% RSLogix 500 project training_bubble_sort_running.RSS, saved by version 8.30.00.16 %
PROJECT "UNTITLED"    % processor: Bul.1763 MicroLogix 1100 Series B %

PROGRAM FILES
  LAD 2 "MAIN"  3 rungs
  LAD 4 "LOADCELLIN"  5 rungs
  LAD 5 "TRAINING"  9 rungs
  LAD 250 "SCANHISTOG"  4 rungs
  LAD 251 "ADD_IRANK6"  7 rungs
  LAD 252 "CALC_PEAKS"  6 rungs
  LAD 253 "RNK6NEWVAL"  6 rungs
  LAD 254 "RNK6BUBBLE"  6 rungs
  LAD 255 "RESETRANK6"  5 rungs

DATA FILES
  O0 OUTPUT  4 elements
  I1 INPUT  6 elements
  S2 STATUS  66 elements
  B3 BINARY  3 elements
  T4 TIMER  2 elements
  C5 COUNTER  1 elements
  R6 CONTROL  1 elements
  N7 INTEGER  66 elements
  F8 FLOAT  1 elements
  L248 SCAN_TIMES  256 elements
  F249 RNK6FLOATS  256 elements
  N250 RNK6_INTS  256 elements
  N251 RNK6COUNTS  7 elements
  N252 RNK6BINS  7 elements
  N253 COUNT_I  256 elements
  N254 RANK6_I  256 elements
  F255 SUM_I  256 elements

LADDER 2 "MAIN"
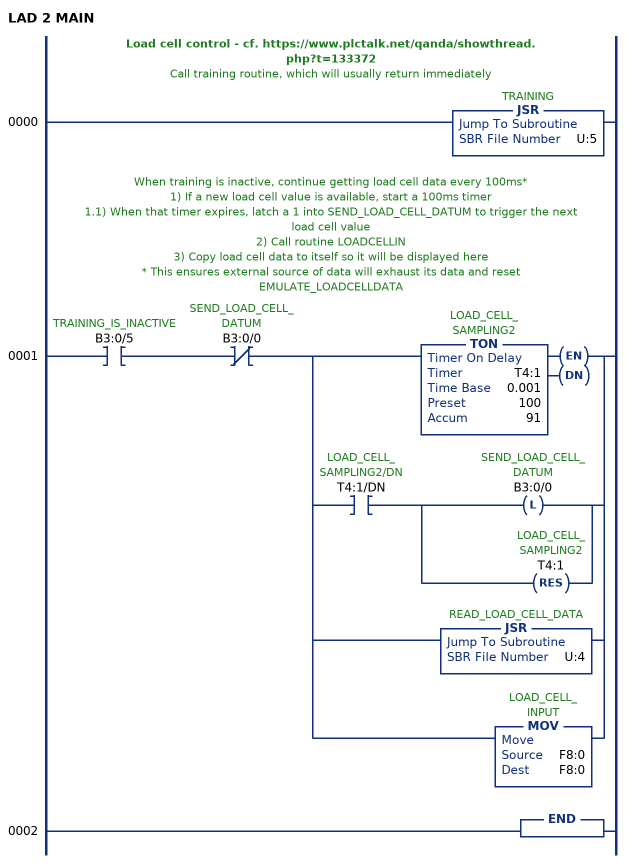
% Rung: 0 %
% TITLE: Load cell control - cf. https://www.plctalk.net/qanda/showthread.php?t=133372 %
% Call training routine, which will usually return immediately %
SOR JSR U:5 EOR
%   U:5  TRAINING %
% Rung: 1 %
% When training is inactive, continue getting load cell data every 100ms*
% 1) If a new load cell value is available, start a 100ms timer
% 1.1) When that timer expires, latch a 1 into SEND_LOAD_CELL_DATUM to trigger the next load cell value
% 2) Call routine LOADCELLIN
% 3) Copy load cell data to itself so it will be displayed here
% * This ensures external source of data will exhaust its data and reset EMULATE_LOADCELLDATA %
SOR XIC B3:0/5 XIO B3:0/0 BST BST TON T4:1 0.001 100 91 NXB XIC T4:1/DN BST OTL B3:0/0 NXB RES T4:1 BND BND NXB JSR U:4 NXB MOV F8:0 F8:0 BND EOR
%   B3:0/5  TRAINING_IS_INACTIVE %
%   B3:0/0  SEND_LOAD_CELL_DATUM %
%   T4:1  LOAD_CELL_SAMPLING2 %
%   U:4  READ_LOAD_CELL_DATA %
%   F8:0  LOAD_CELL_INPUT %
% Rung: 2 %
SOR END EOR

LADDER 4 "LOADCELLIN"
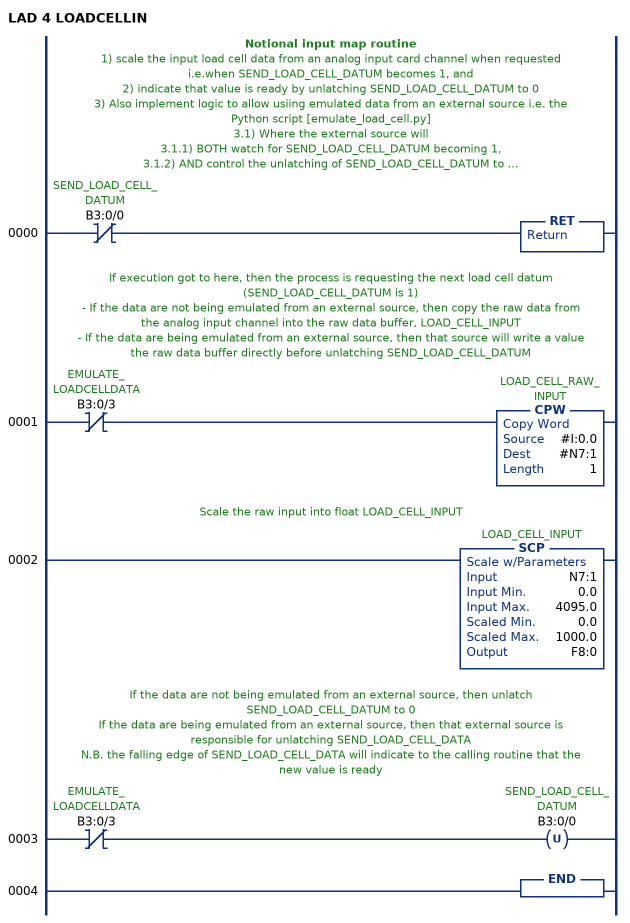
% Rung: 0 %
% TITLE: Notional input map routine %
% 1) scale the input load cell data from an analog input card channel when requested i.e.when SEND_LOAD_CELL_DATUM becomes 1, and
% 2) indicate that value is ready by unlatching SEND_LOAD_CELL_DATUM to 0
% 3) Also implement logic to allow usiing emulated data from an external source i.e. the Python script [emulate_load_cell.py]
% 3.1) Where the external source will
% 3.1.1) BOTH watch for SEND_LOAD_CELL_DATUM becoming 1,
% 3.1.2) AND control the unlatching of SEND_LOAD_CELL_DATUM to 0
% 
% ========================================================================
% If SEND_LOAD_CELL_DATA is 0 i.e. not 1, then return and do nothing %
SOR XIO B3:0/0 RET EOR
%   B3:0/0  SEND_LOAD_CELL_DATUM %
% Rung: 1 %
% If execution got to here, then the process is requesting the next load cell datum (SEND_LOAD_CELL_DATUM is 1)
% - If the data are not being emulated from an external source, then copy the raw data from the analog input channel into the raw data buffer, LOAD_CELL_INPUT
% - If the data are being emulated from an external source, then that source will write a value the raw data buffer directly before unlatching SEND_LOAD_CELL_DATUM %
SOR XIO B3:0/3 CPW #I:0.0 #N7:1 1 EOR
%   B3:0/3  EMULATE_LOADCELLDATA %
%   N7:1  LOAD_CELL_RAW_INPUT %
% Rung: 2 %
% Scale the raw input into float LOAD_CELL_INPUT %
SOR SCP N7:1 0.0 4095.0 0.0 1000.0 F8:0 EOR
%   N7:1  LOAD_CELL_RAW_INPUT %
%   F8:0  LOAD_CELL_INPUT %
% Rung: 3 %
% If the data are not being emulated from an external source, then unlatch SEND_LOAD_CELL_DATUM to 0
% If the data are being emulated from an external source, then that external source is responsible for unlatching SEND_LOAD_CELL_DATA
% N.B. the falling edge of SEND_LOAD_CELL_DATA will indicate to the calling routine that the new value is ready %
SOR XIO B3:0/3 OTU B3:0/0 EOR
%   B3:0/3  EMULATE_LOADCELLDATA %
%   B3:0/0  SEND_LOAD_CELL_DATUM %
% Rung: 4 %
SOR END EOR

LADDER 5 "TRAINING"
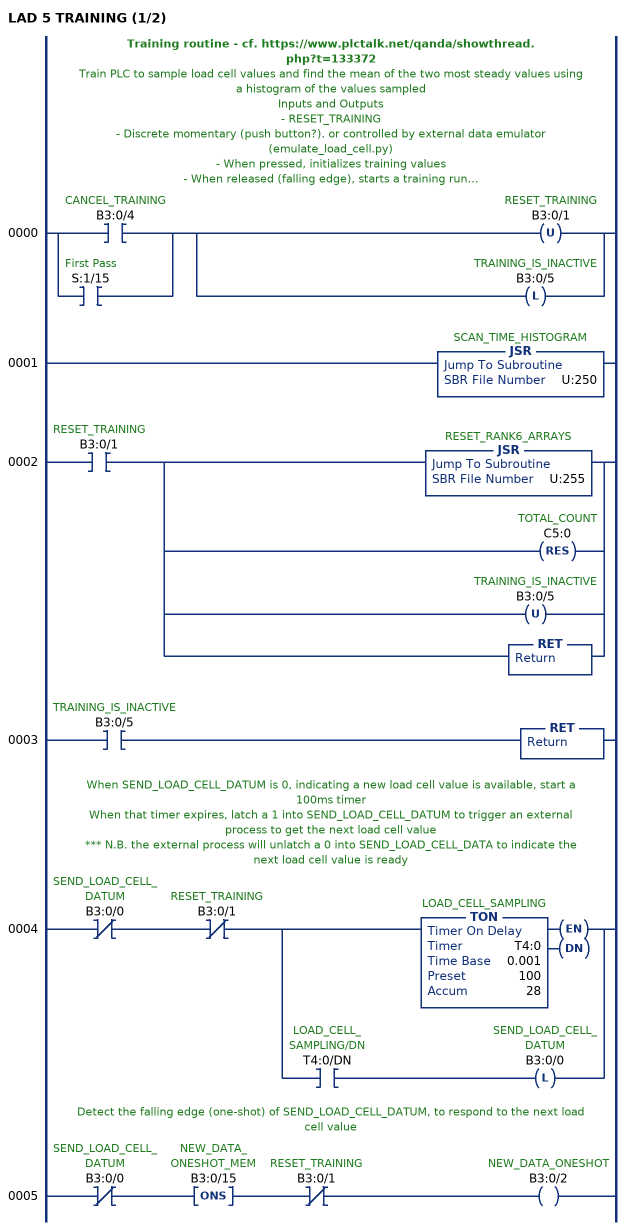
% Rung: 0 %
% TITLE: Training routine - cf. https://www.plctalk.net/qanda/showthread.php?t=133372 %
% Train PLC to sample load cell values and find the mean of the two most steady values using
% a histogram of the values sampled
% 
% Inputs and Outputs
% - RESET_TRAINING
%   - Discrete momentary (push button?). or controlled by external data emulator (emulate_load_cell.py)
%   - When pressed, initializes training values
%   - When released (falling edge), starts a training rung
% - LOAD_CELL_INPUT
%   - Analog float value that is loaded from load cell in response to a rising edge of Boolean SEND_LOAD_CELL_DATUM
% - SEND_LOAD_CELL_DATUM (both output-ish and input-ish)
%   - Output:  written to as a 1 by this routine to indicate 100ms have expired and it is time for the next load cell value
%   - Input:  written to as a 0 by another entity to after putting a new value into LOAD_CELL_INPUT
%     - This falling edge indicates a new LOAD_CELL_INPUT is ready
%     - The other entity could be an I/O mapping routine, or the Python script [emulate_load_cell.py]
% 
% ========================================================================
% First rung:  respond to request to cancel training %
SOR BST XIC B3:0/4 NXB XIC S:1/15 BND BST OTU B3:0/1 NXB OTL B3:0/5 BND EOR
%   B3:0/4  CANCEL_TRAINING %
%   S:1/15  "First Pass" %
%   B3:0/1  RESET_TRAINING %
%   B3:0/5  TRAINING_IS_INACTIVE %
% Rung: 1 %
SOR JSR U:250 EOR
%   U:250  SCAN_TIME_HISTOGRAM %
% Rung: 2 %
SOR XIC B3:0/1 BST JSR U:255 NXB RES C5:0 NXB OTU B3:0/5 NXB RET BND EOR
%   B3:0/1  RESET_TRAINING %
%   U:255  RESET_RANK6_ARRAYS %
%   C5:0  TOTAL_COUNT %
%   B3:0/5  TRAINING_IS_INACTIVE %
% Rung: 3 %
SOR XIC B3:0/5 RET EOR
%   B3:0/5  TRAINING_IS_INACTIVE %
% Rung: 4 %
% When SEND_LOAD_CELL_DATUM is 0, indicating a new load cell value is available, start a 100ms timer
% When that timer expires, latch a 1 into SEND_LOAD_CELL_DATUM to trigger an external process to get the next load cell value
% *** N.B. the external process will unlatch a 0 into SEND_LOAD_CELL_DATA to indicate the next load cell value is ready %
SOR XIO B3:0/0 XIO B3:0/1 BST TON T4:0 0.001 100 28 NXB XIC T4:0/DN OTL B3:0/0 BND EOR
%   B3:0/0  SEND_LOAD_CELL_DATUM %
%   B3:0/1  RESET_TRAINING %
%   T4:0  LOAD_CELL_SAMPLING %
% Rung: 5 %
% Detect the falling edge (one-shot) of SEND_LOAD_CELL_DATUM, to respond to the next load cell value %
SOR XIO B3:0/0 ONS B3:0/15 XIO B3:0/1 OTE B3:0/2 EOR
%   B3:0/0  SEND_LOAD_CELL_DATUM %
%   B3:0/15  NEW_DATA_ONESHOT_MEM %
%   B3:0/1  RESET_TRAINING %
%   B3:0/2  NEW_DATA_ONESHOT %

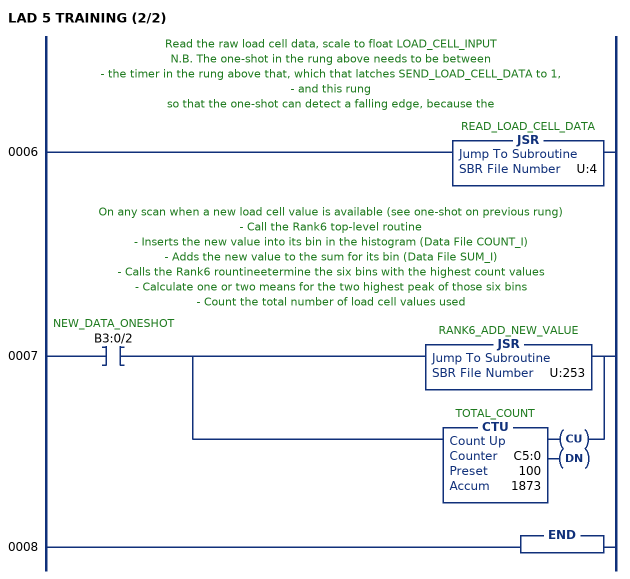
% Rung: 6 %
% Read the raw load cell data, scale to float LOAD_CELL_INPUT
% 
% N.B. The one-shot in the rung above needs to be between
%         - the timer in the rung above that, which that latches SEND_LOAD_CELL_DATA to 1,
%         - and this rung
%         so that the one-shot can detect a falling edge, because the %
SOR JSR U:4 EOR
%   U:4  READ_LOAD_CELL_DATA %
% Rung: 7 %
% On any scan when a new load cell value is available (see one-shot on previous rung)
% - Call the Rank6 top-level routine
%   - Inserts the new value into its bin in the histogram (Data File COUNT_I)
%   - Adds the new value to the sum for its bin (Data File SUM_I)
%   - Calls the Rank6 rountineetermine the six bins with the highest count values
%   - Calculate one or two means for the two highest peak of those six bins
% - Count the total number of load cell values used %
SOR XIC B3:0/2 BST JSR U:253 NXB CTU C5:0 100 1873 BND EOR
%   B3:0/2  NEW_DATA_ONESHOT %
%   U:253  RANK6_ADD_NEW_VALUE %
%   C5:0  TOTAL_COUNT %
% Rung: 8 %
SOR END EOR

LADDER 250 "SCANHISTOG"
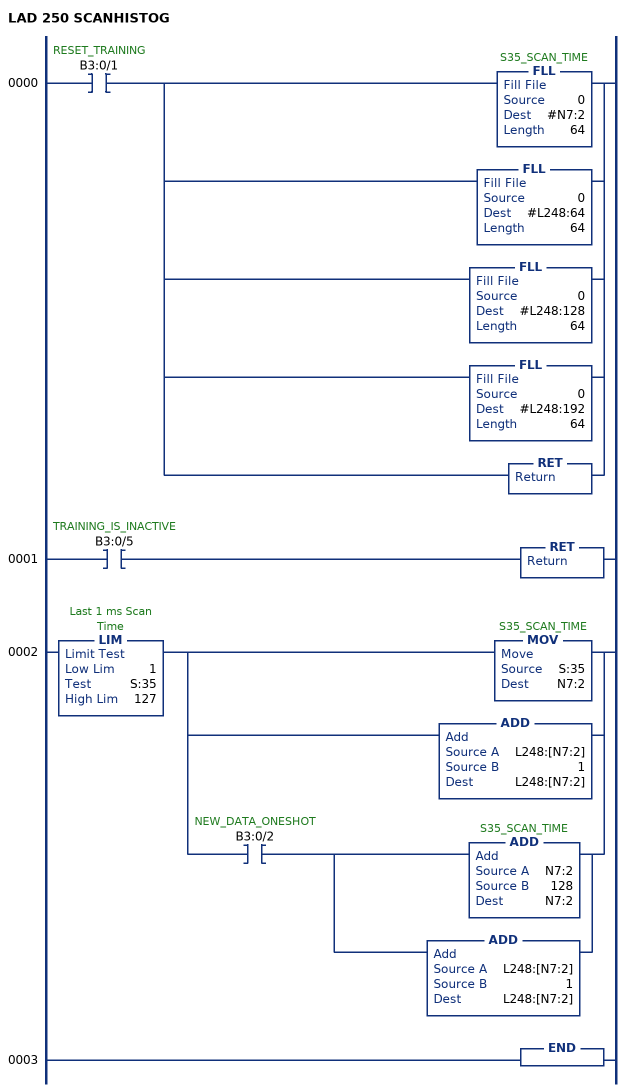
% Rung: 0 %
SOR XIC B3:0/1 BST FLL 0 #N7:2 64 NXB FLL 0 #L248:64 64 NXB FLL 0 #L248:128 64 NXB FLL 0 #L248:192 64 NXB RET BND EOR
%   B3:0/1  RESET_TRAINING %
%   N7:2  S35_SCAN_TIME %
% Rung: 1 %
SOR XIC B3:0/5 RET EOR
%   B3:0/5  TRAINING_IS_INACTIVE %
% Rung: 2 %
SOR LIM 1 S:35 127 BST MOV S:35 N7:2 NXB ADD L248:[N7:2] 1 L248:[N7:2] NXB XIC B3:0/2 BST ADD N7:2 128 N7:2 NXB ADD L248:[N7:2] 1 L248:[N7:2] BND BND EOR
%   S:35  "Last 1 ms Scan Time" %
%   N7:2  S35_SCAN_TIME %
%   B3:0/2  NEW_DATA_ONESHOT %
% Rung: 3 %
SOR END EOR

LADDER 251 "ADD_IRANK6"
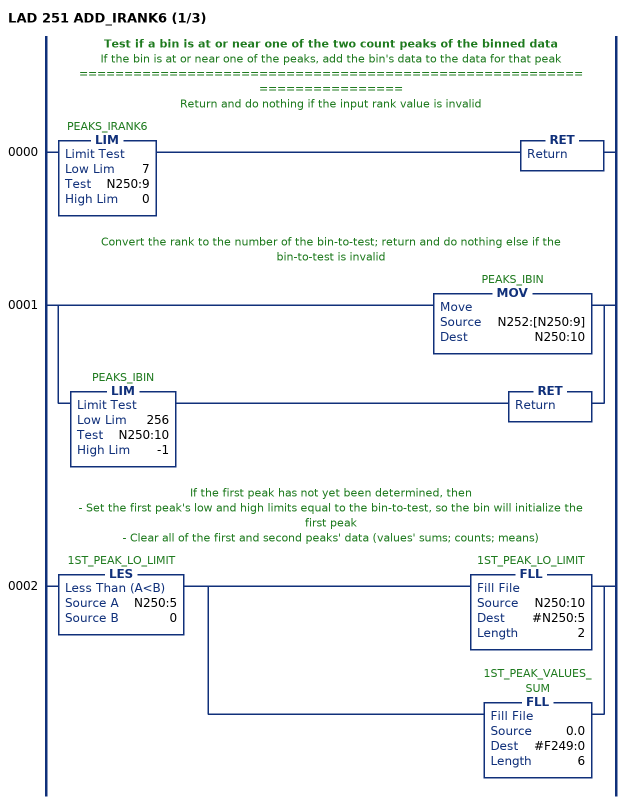
% Rung: 0 %
% TITLE: Test if a bin is at or near one of the two count peaks of the binned data %
% If the bin is at or near one of the peaks, add the bin's data to the data for that peak
% 
% ========================================================================
% Return and do nothing if the input rank value is invalid %
SOR LIM 7 N250:9 0 RET EOR
%   N250:9  PEAKS_IRANK6 %
% Rung: 1 %
% Convert the rank to the number of the bin-to-test; return and do nothing else if the bin-to-test is invalid %
SOR BST MOV N252:[N250:9] N250:10 NXB LIM 256 N250:10 -1 RET BND EOR
%   N250:9  PEAKS_IRANK6 %
%   N250:10  PEAKS_IBIN %
% Rung: 2 %
% If the first peak has not yet been determined, then
% - Set the first peak's low and high limits equal to the bin-to-test, so the bin will initialize the first peak
% - Clear all of the first and second peaks' data (values' sums; counts; means) %
SOR LES N250:5 0 BST FLL N250:10 #N250:5 2 NXB FLL 0.0 #F249:0 6 BND EOR
%   N250:5  1ST_PEAK_LO_LIMIT %
%   N250:10  PEAKS_IBIN %
%   F249:0  1ST_PEAK_VALUES_SUM %

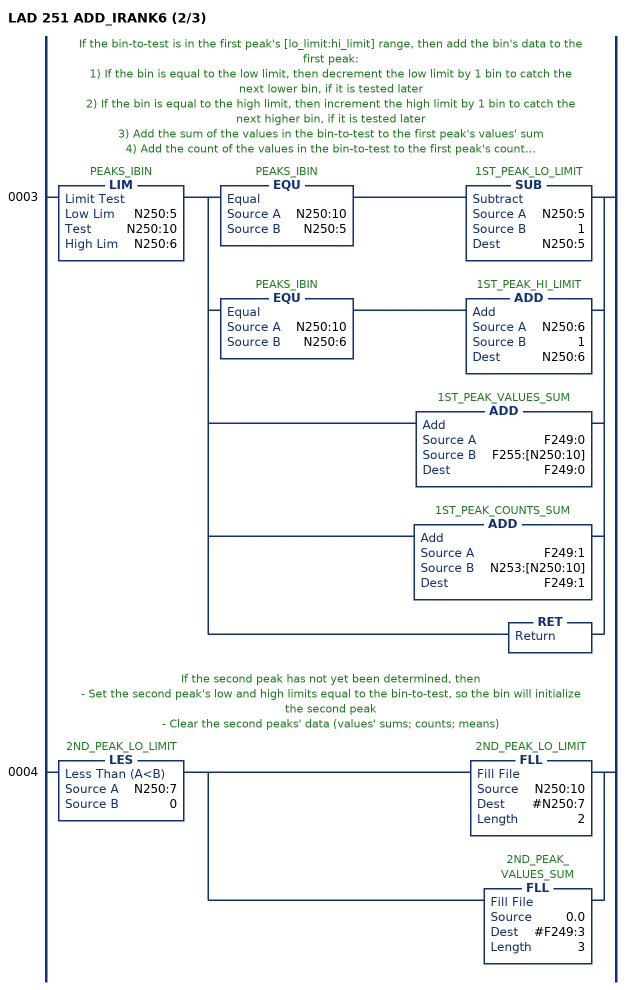
% Rung: 3 %
% If the bin-to-test is in the first peak's [lo_limit:hi_limit] range, then add the bin's data to the first peak:
% 1) If the bin is equal to the low limit, then decrement the low limit by 1 bin to catch the next lower bin, if it is tested later
% 2) If the bin is equal to the high limit, then increment the high limit by 1 bin to catch the next higher bin, if it is tested later
% 3) Add the sum of the values in the bin-to-test to the first peak's values' sum
% 4) Add the count of the values in the bin-to-test to the first peak's counts
% 5) Return and do nothing else in this routine, because the bin-to-test is in the first peak, so it cannot be in the second peak %
SOR LIM N250:5 N250:10 N250:6 BST EQU N250:10 N250:5 SUB N250:5 1 N250:5 NXB EQU N250:10 N250:6 ADD N250:6 1 N250:6 NXB ADD F249:0 F255:[N250:10] F249:0 NXB ADD F249:1 N253:[N250:10] F249:1 NXB RET BND EOR
%   N250:5  1ST_PEAK_LO_LIMIT %
%   N250:10  PEAKS_IBIN %
%   N250:6  1ST_PEAK_HI_LIMIT %
%   F249:0  1ST_PEAK_VALUES_SUM %
%   F249:1  1ST_PEAK_COUNTS_SUM %
% Rung: 4 %
% If the second peak has not yet been determined, then
% - Set the second peak's low and high limits equal to the bin-to-test, so the bin will initialize the second peak
% - Clear the second peaks' data (values' sums; counts; means) %
SOR LES N250:7 0 BST FLL N250:10 #N250:7 2 NXB FLL 0.0 #F249:3 3 BND EOR
%   N250:7  2ND_PEAK_LO_LIMIT %
%   N250:10  PEAKS_IBIN %
%   F249:3  2ND_PEAK_VALUES_SUM %

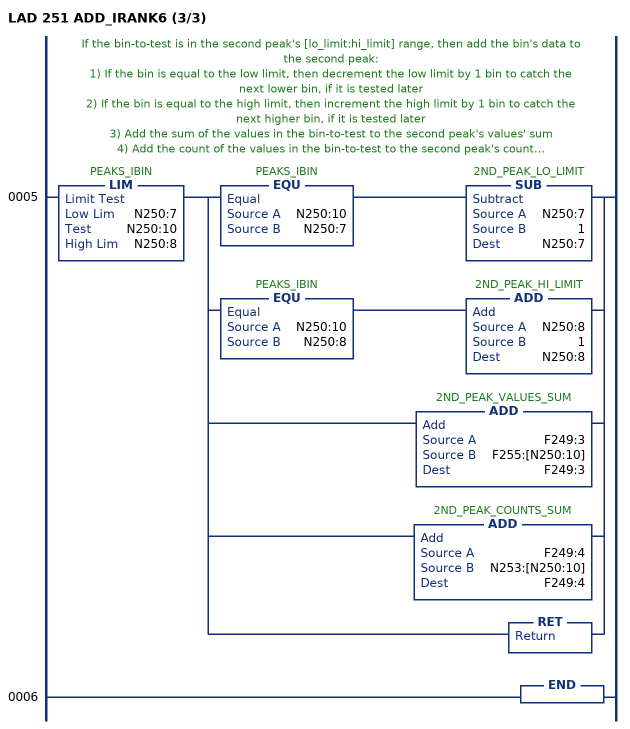
% Rung: 5 %
% If the bin-to-test is in the second peak's [lo_limit:hi_limit] range, then add the bin's data to the second peak:
% 1) If the bin is equal to the low limit, then decrement the low limit by 1 bin to catch the next lower bin, if it is tested later
% 2) If the bin is equal to the high limit, then increment the high limit by 1 bin to catch the next higher bin, if it is tested later
% 3) Add the sum of the values in the bin-to-test to the second peak's values' sum
% 4) Add the count of the values in the bin-to-test to the second peak's counts
% 5) The return is superfluous since this was originally the last rung in this routine, but this leaves open the possibility to add more peaks %
SOR LIM N250:7 N250:10 N250:8 BST EQU N250:10 N250:7 SUB N250:7 1 N250:7 NXB EQU N250:10 N250:8 ADD N250:8 1 N250:8 NXB ADD F249:3 F255:[N250:10] F249:3 NXB ADD F249:4 N253:[N250:10] F249:4 NXB RET BND EOR
%   N250:7  2ND_PEAK_LO_LIMIT %
%   N250:10  PEAKS_IBIN %
%   N250:8  2ND_PEAK_HI_LIMIT %
%   F249:3  2ND_PEAK_VALUES_SUM %
%   F249:4  2ND_PEAK_COUNTS_SUM %
% Rung: 6 %
SOR END EOR

LADDER 252 "CALC_PEAKS"
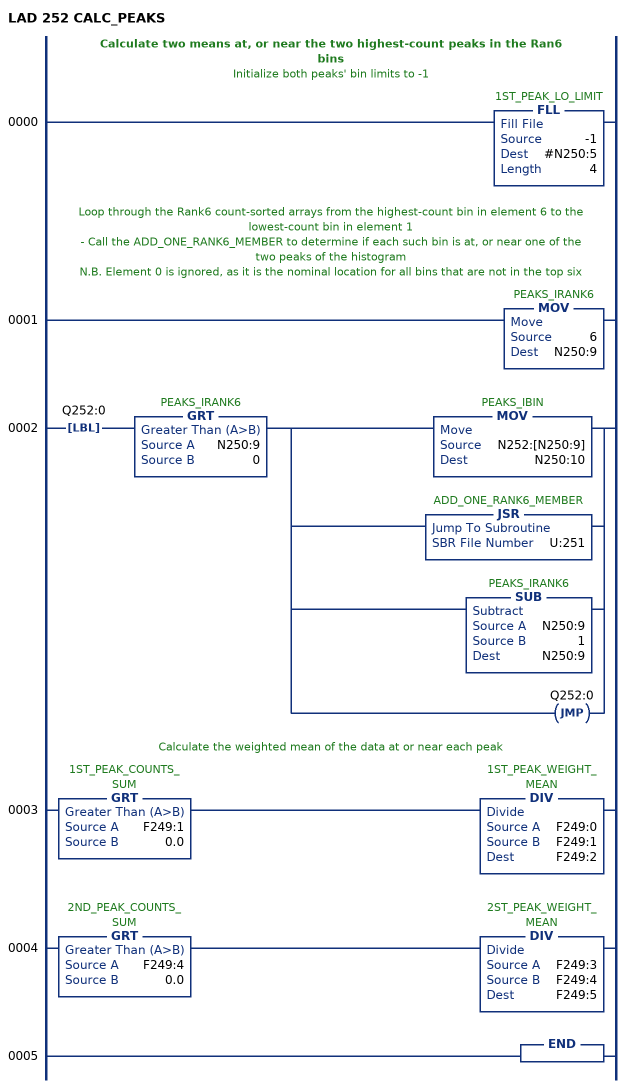
% Rung: 0 %
% TITLE: Calculate two means at, or near the two highest-count peaks in the Ran6 bins %
% Initialize both peaks' bin limits to -1 %
SOR FLL -1 #N250:5 4 EOR
%   N250:5  1ST_PEAK_LO_LIMIT %
% Rung: 1 %
% Loop through the Rank6 count-sorted arrays from the highest-count bin in element 6 to the lowest-count bin in element 1
% - Call the ADD_ONE_RANK6_MEMBER to determine if each such bin is at, or near one of the two peaks of the histogram
% N.B. Element 0 is ignored, as it is the nominal location for all bins that are not in the top six %
SOR MOV 6 N250:9 EOR
%   N250:9  PEAKS_IRANK6 %
% Rung: 2 %
SOR LBL Q252:0 GRT N250:9 0 BST MOV N252:[N250:9] N250:10 NXB JSR U:251 NXB SUB N250:9 1 N250:9 NXB JMP Q252:0 BND EOR
%   N250:9  PEAKS_IRANK6 %
%   N250:10  PEAKS_IBIN %
%   U:251  ADD_ONE_RANK6_MEMBER %
% Rung: 3 %
% Calculate the weighted mean of the data at or near each peak %
SOR GRT F249:1 0.0 DIV F249:0 F249:1 F249:2 EOR
%   F249:1  1ST_PEAK_COUNTS_SUM %
%   F249:0  1ST_PEAK_VALUES_SUM %
%   F249:2  1ST_PEAK_WEIGHT_MEAN %
% Rung: 4 %
SOR GRT F249:4 0.0 DIV F249:3 F249:4 F249:5 EOR
%   F249:4  2ND_PEAK_COUNTS_SUM %
%   F249:3  2ND_PEAK_VALUES_SUM %
%   F249:5  2ST_PEAK_WEIGHT_MEAN %
% Rung: 5 %
SOR END EOR

LADDER 253 "RNK6NEWVAL"
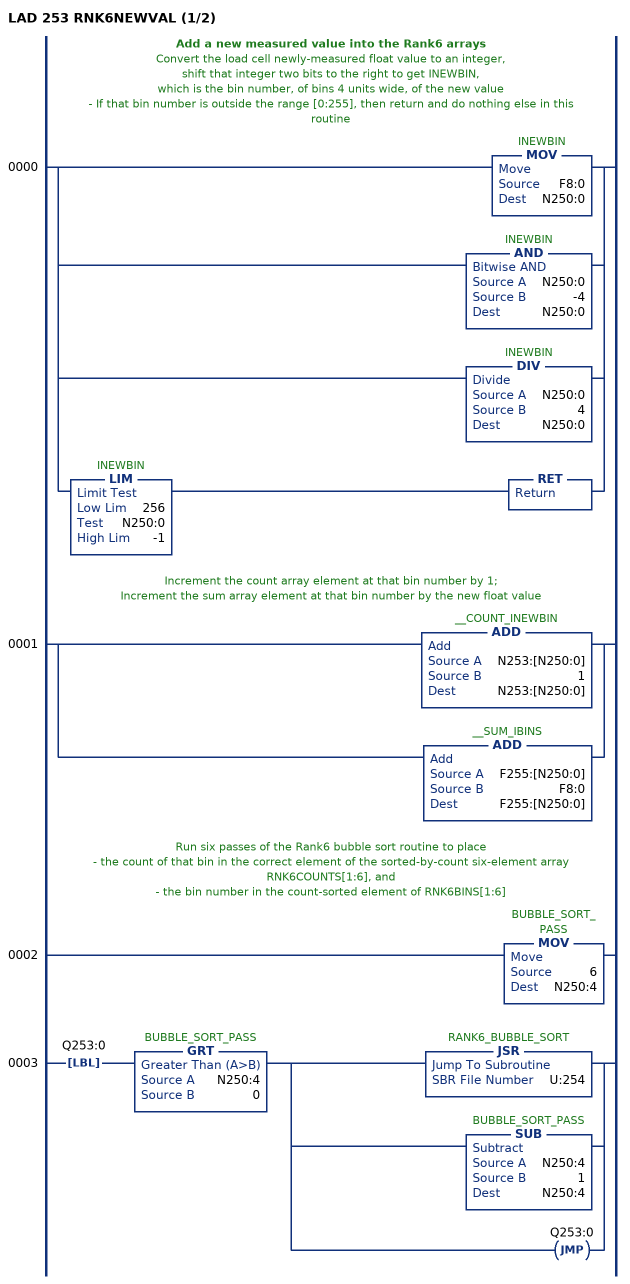
% Rung: 0 %
% TITLE: Add a new measured value into the Rank6 arrays %
% Convert the load cell newly-measured float value to an integer,
% shift that integer two bits to the right to get INEWBIN,
% which is the bin number, of bins 4 units wide, of the new value
% - If that bin number is outside the range [0:255], then return and do nothing else in this routine %
SOR BST MOV F8:0 N250:0 NXB AND N250:0 -4 N250:0 NXB DIV N250:0 4 N250:0 NXB LIM 256 N250:0 -1 RET BND EOR
%   F8:0  LOAD_CELL_INPUT %
%   N250:0  INEWBIN %
% Rung: 1 %
% Increment the count array element at that bin number by 1;
% Increment the sum array element at that bin number by the new float value %
SOR BST ADD N253:[N250:0] 1 N253:[N250:0] NXB ADD F255:[N250:0] F8:0 F255:[N250:0] BND EOR
%   N253:[N250:0]  __COUNT_INEWBIN %
%   N250:0  INEWBIN %
%   F255:[N250:0]  __SUM_IBINS %
%   F8:0  LOAD_CELL_INPUT %
% Rung: 2 %
% Run six passes of the Rank6 bubble sort routine to place
% - the count of that bin in the correct element of the sorted-by-count six-element array RNK6COUNTS[1:6], and
% - the bin number in the count-sorted element of RNK6BINS[1:6] %
SOR MOV 6 N250:4 EOR
%   N250:4  BUBBLE_SORT_PASS %
% Rung: 3 %
SOR LBL Q253:0 GRT N250:4 0 BST JSR U:254 NXB SUB N250:4 1 N250:4 NXB JMP Q253:0 BND EOR
%   N250:4  BUBBLE_SORT_PASS %
%   U:254  RANK6_BUBBLE_SORT %

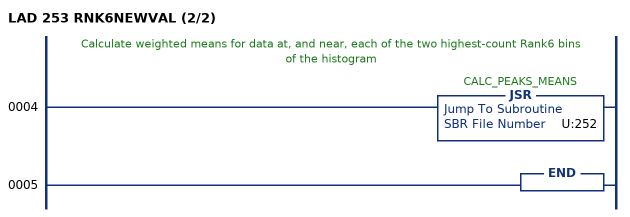
% Rung: 4 %
% Calculate weighted means for data at, and near, each of the two highest-count Rank6 bins of the histogram %
SOR JSR U:252 EOR
%   U:252  CALC_PEAKS_MEANS %
% Rung: 5 %
SOR END EOR

LADDER 254 "RNK6BUBBLE"
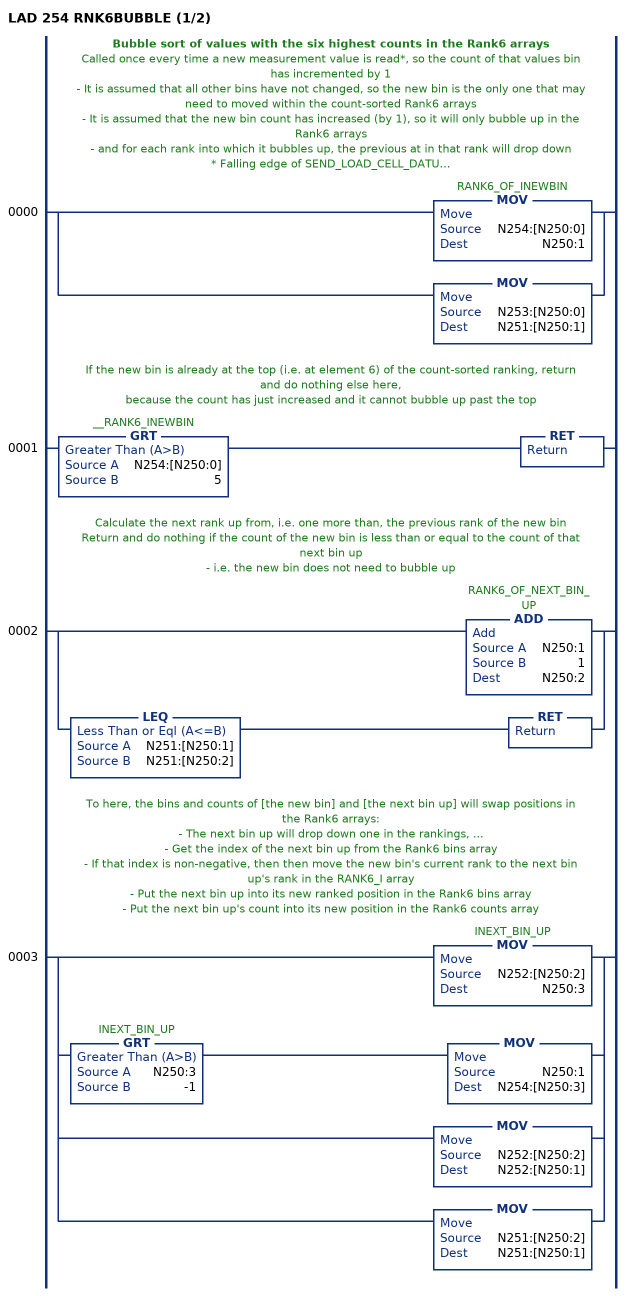
% Rung: 0 %
% TITLE: Bubble sort of values with the six highest counts in the Rank6 arrays %
% Called once every time a new measurement value is read*, so the count of that values bin has incremented by 1
% - It is assumed that all other bins have not changed, so the new bin is the only one that may need to moved within the count-sorted Rank6 arrays
% - It is assumed that the new bin count has increased (by 1), so it will only bubble up in the Rank6 arrays
%   - and for each rank into which it bubbles up, the previous at in that rank will drop down
% 
% * Falling edge of SEND_LOAD_CELL_DATUM
% 
% ========================================================================
% Get current rank of the new bin from the Rank6 bins array
% Place the updated count of the new bin in the ranked position of that bin in the Rank6 counts array %
SOR BST MOV N254:[N250:0] N250:1 NXB MOV N253:[N250:0] N251:[N250:1] BND EOR
%   N254:[N250:0]  __RANK6_INEWBIN %
%   N250:0  INEWBIN %
%   N250:1  RANK6_OF_INEWBIN %
%   N253:[N250:0]  __COUNT_INEWBIN %
% Rung: 1 %
% If the new bin is already at the top (i.e. at element 6) of the count-sorted ranking, return and do nothing else here,
% because the count has just increased and it cannot bubble up past the top %
SOR GRT N254:[N250:0] 5 RET EOR
%   N254:[N250:0]  __RANK6_INEWBIN %
%   N250:0  INEWBIN %
% Rung: 2 %
% Calculate the next rank up from, i.e. one more than, the previous rank of the new bin
% Return and do nothing if the count of the new bin is less than or equal to the count of that next bin up
% - i.e. the new bin does not need to bubble up %
SOR BST ADD N250:1 1 N250:2 NXB LEQ N251:[N250:1] N251:[N250:2] RET BND EOR
%   N250:1  RANK6_OF_INEWBIN %
%   N250:2  RANK6_OF_NEXT_BIN_UP %
% Rung: 3 %
% To here, the bins and counts of [the new bin] and [the next bin up] will swap positions in the Rank6 arrays:
% - The next bin up will drop down one in the rankings, ...
%   - Get the index of the next bin up from the Rank6 bins array
%   - If that index is non-negative, then then move the new bin's current rank to the next bin up's rank in the RANK6_I array
%   - Put the next bin up into its new ranked position in the Rank6 bins array
%   - Put the next bin up's count into its new position in the Rank6 counts array %
SOR BST MOV N252:[N250:2] N250:3 NXB GRT N250:3 -1 MOV N250:1 N254:[N250:3] NXB MOV N252:[N250:2] N252:[N250:1] NXB MOV N251:[N250:2] N251:[N250:1] BND EOR
%   N250:2  RANK6_OF_NEXT_BIN_UP %
%   N250:3  INEXT_BIN_UP %
%   N250:1  RANK6_OF_INEWBIN %

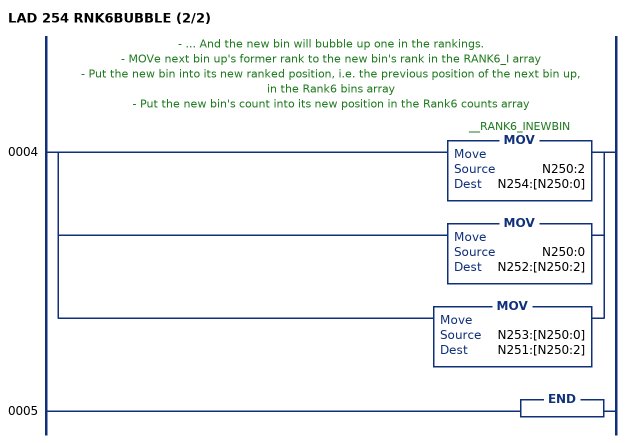
% Rung: 4 %
% - ... And the new bin will bubble up one in the rankings.
%   - MOVe next bin up's former rank to the new bin's rank in the RANK6_I array
%   - Put the new bin into its new ranked position, i.e. the previous position of the next bin up, in the Rank6 bins array
%   - Put the new bin's count into its new position in the Rank6 counts array %
SOR BST MOV N250:2 N254:[N250:0] NXB MOV N250:0 N252:[N250:2] NXB MOV N253:[N250:0] N251:[N250:2] BND EOR
%   N250:2  RANK6_OF_NEXT_BIN_UP %
%   N254:[N250:0]  __RANK6_INEWBIN %
%   N250:0  INEWBIN %
%   N253:[N250:0]  __COUNT_INEWBIN %
% Rung: 5 %
SOR END EOR

LADDER 255 "RESETRANK6"
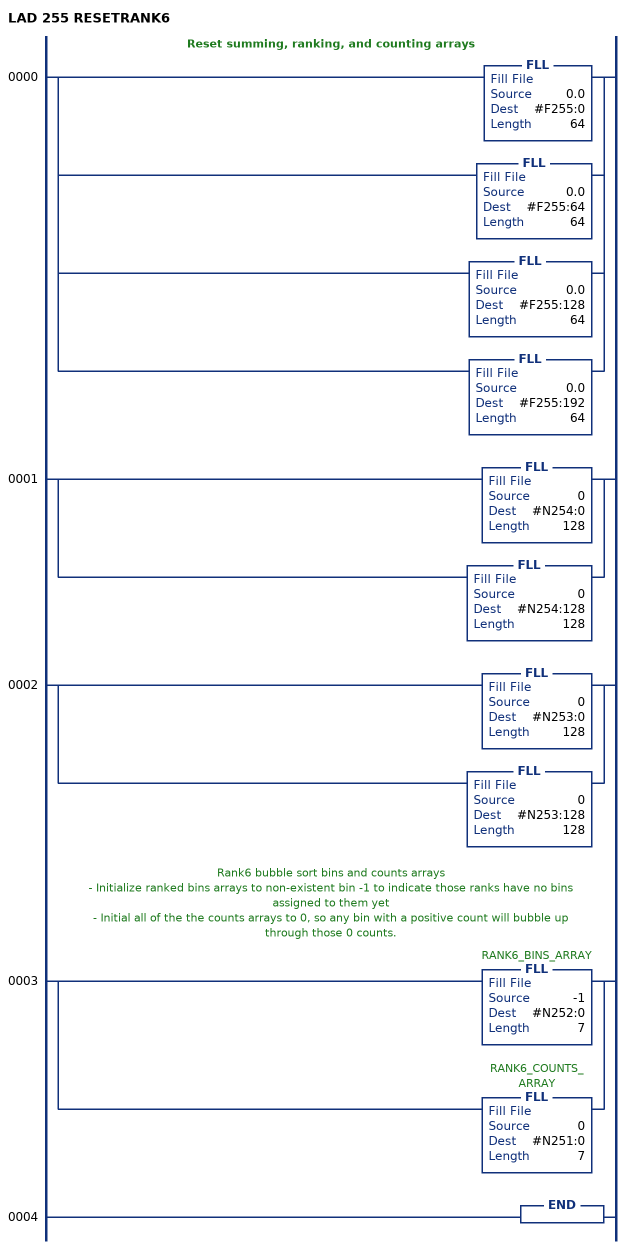
% Rung: 0 %
% TITLE: Reset summing, ranking, and counting arrays %
SOR BST FLL 0.0 #F255:0 64 NXB FLL 0.0 #F255:64 64 NXB FLL 0.0 #F255:128 64 NXB FLL 0.0 #F255:192 64 BND EOR
% Rung: 1 %
SOR BST FLL 0 #N254:0 128 NXB FLL 0 #N254:128 128 BND EOR
% Rung: 2 %
SOR BST FLL 0 #N253:0 128 NXB FLL 0 #N253:128 128 BND EOR
% Rung: 3 %
% Rank6 bubble sort bins and counts arrays
% - Initialize ranked bins arrays to non-existent bin -1 to indicate those ranks have no bins assigned to them yet
% - Initial all of the the counts arrays to 0, so any bin with a positive count will bubble up through those 0 counts. %
SOR BST FLL -1 #N252:0 7 NXB FLL 0 #N251:0 7 BND EOR
%   N252:0  RANK6_BINS_ARRAY %
%   N251:0  RANK6_COUNTS_ARRAY %
% Rung: 4 %
SOR END EOR

OTHER DOCUMENTED ADDRESSES
  B3:0/6  TRAINING_FINISHED
  B3:0/13  TRAINING_FINISH_ONSM
  B3:0/14  RESET_FALLING_ONS_M
  F8:1  FILTERED_DATA
  F8:2  FILTER_PARAMETER
  F8:3  TEMPORARY_FLOAT
  F8:4  DATA_DIFFERENCE
  F8:5  FILTERED_DATA_LOW
  F8:6  FILTERED_DATA_HIGH
  F8:7  FILTERED_DATA_THIRD
  N7:0  PASS_NUMBER
  U:3  FILTER_DATA

COMMENTS NOT ATTACHED TO A CURRENT RUNG
  T4:0: Initialize and set up for training run

DATA TABLE (non-zero values as saved)
DATA B3
% B3:0 % 0X8020 0X0000 0X0000
DATA T4
% .PRE .ACC %
% T4:0 % 100 28
% T4:1 % 100 91
DATA C5
% .PRE .ACC %
% C5:0 % 100 1873
DATA R6
% .LEN .POS %
% R6:0 % 16 0
DATA N7
% N7:0 % 0 0 6 0 0 0 0 0 0 0
DATA L248
% L248:5 % 0 38767 92330 46761 14472
% L248:10 % 24269 23135 18152 10832 5463
% L248:15 % 4244 4354 3832 2332 1206
% L248:20 % 604 479 475 398 293
% L248:25 % 294 287 202 151 107
% L248:30 % 57 77 95 77 37
% L248:35 % 9 8 21 22 16
% L248:40 % 11 4 2 2 2
% L248:45 % 1 7 47 108 242
% L248:50 % 176 118 77 100 137
% L248:55 % 176 168 98 54 28
% L248:60 % 7 18 9 8 7
% L248:65 % 11 10 9 1 1
% L248:70 % 1 1 2 1 0
% L248:155 % 0 0 0 0 19
% L248:160 % 49 59 31 6 6
% L248:165 % 21 22 16 11 4
% L248:170 % 2 2 2 1 7
% L248:175 % 47 108 242 176 118
% L248:180 % 77 100 137 176 168
% L248:185 % 98 54 28 7 18
% L248:190 % 9 8 7 11 10
% L248:195 % 9 1 1 1 1
% L248:200 % 2 1 0 0 0
DATA F249
% F249:0 % 252297.8 931 270.9966 106421.1 579
% F249:5 % 183.8016 0 0 0 0
DATA N250
% N250:0 % 46 5 6 68 0 66 70 44 47 0
% N250:10 % 38 0 0 0 0 0 0 0 0 0
DATA N251
% N251:0 % 19 39 39 234 329 345 563
DATA N252
% N252:0 % 70 38 69 45 68 46 67
DATA N253
% N253:20 % 0 0 0 0 0 0 0 0 5 4
% N253:30 % 7 6 9 23 18 10 4 12 39 9
% N253:40 % 5 1 3 3 19 234 345 15 6 2
% N253:50 % 4 2 7 5 4 4 3 3 2 1
% N253:60 % 5 6 4 7 4 10 19 563 329 39
% N253:70 % 34 4 0 1 2 1 2 0 3 4
% N253:80 % 1 1 0 0 1 0 0 0 1 0
% N253:90 % 1 1 0 1 0 0 1 0 0 1
% N253:100 % 0 1 0 0 1 2 0 2 2 2
% N253:110 % 1 2 0 0 0 0 0 0 0 0
DATA N254
% N254:30 % 0 0 0 0 0 0 0 0 1 0
% N254:40 % 0 0 0 0 0 3 5 0 0 0
% N254:60 % 0 0 0 0 0 0 0 6 4 2
DATA F255
% F255:25 % 0 0 0 572.8938 468.8645
% F255:30 % 849.0842 749.6947 1161.416 3073.26 2471.795
% F255:35 % 1410.745 586.3248 1799.267 5978.022 1417.582
% F255:40 % 803.4188 164.1026 506.2271 522.3444 3364.103
% F255:45 % 42745.34 63675.77 2842.735 1157.753 394.1392
% F255:50 % 803.663 409.5238 1466.178 1068.62 867.3993
% F255:55 % 884.7375 676.1905 688.4005 468.8645 237.1184
% F255:60 % 1205.861 1475.214 994.3834 1772.161 1028.083
% F255:65 % 2613.187 5060.317 151760.3 89690.55 10846.88
% F255:70 % 9528.692 1146.276 0 295.2381 594.3834
% F255:75 % 300.6105 608.7912 0 938.7057 1269.841
% F255:80 % 320.1465 325.0305 0 0 338.4615
% F255:85 % 0 0 0 351.6483 0
% F255:90 % 361.4164 364.3468 0 373.138 0
% F255:95 % 0 386.0806 0 0 395.6044
% F255:100 % 0 405.8608 0 0 417.3382
% F255:105 % 843.7119 0 859.3407 867.6434 874.9695
% F255:110 % 441.514 888.6447 0 0 0
